(* PLC project Unnamed, Unknown Unnamed 1 *)
(* stored: creationDateTime 2023-10-18T21:45:43, modificationDateTime 2023-10-21T23:16:36 *)

PROGRAM program0
  VAR
    Emrg_Stop : BOOL;
    Output_switch : BOOL;
    change_filter : BOOL;
    Gray_water_level : INT;
    Filter_Input_water_level : INT;
    Filter_Output_water_level : INT;
    Clean_water_level : INT := 0;
    Graywater_Pump_RPM : INT;
    Filterwater_Pump_RPM : INT;
    Cleanwater_Pump_RPM : INT;
    Filterwater_Valve : BOOL;
    Cleanwater_Valve : BOOL;
    Filter_inflow_Valve : BOOL;
    Min_Water_Level : INT := 5;
    Max_Water_Level : INT := 25;
    Max_pump_speed : INT := 2000;
    Min_pump_speed : INT := 0;
    Mem1 : BOOL;
    Mem2 : BOOL;
    Mem3 : BOOL;
  END_VAR

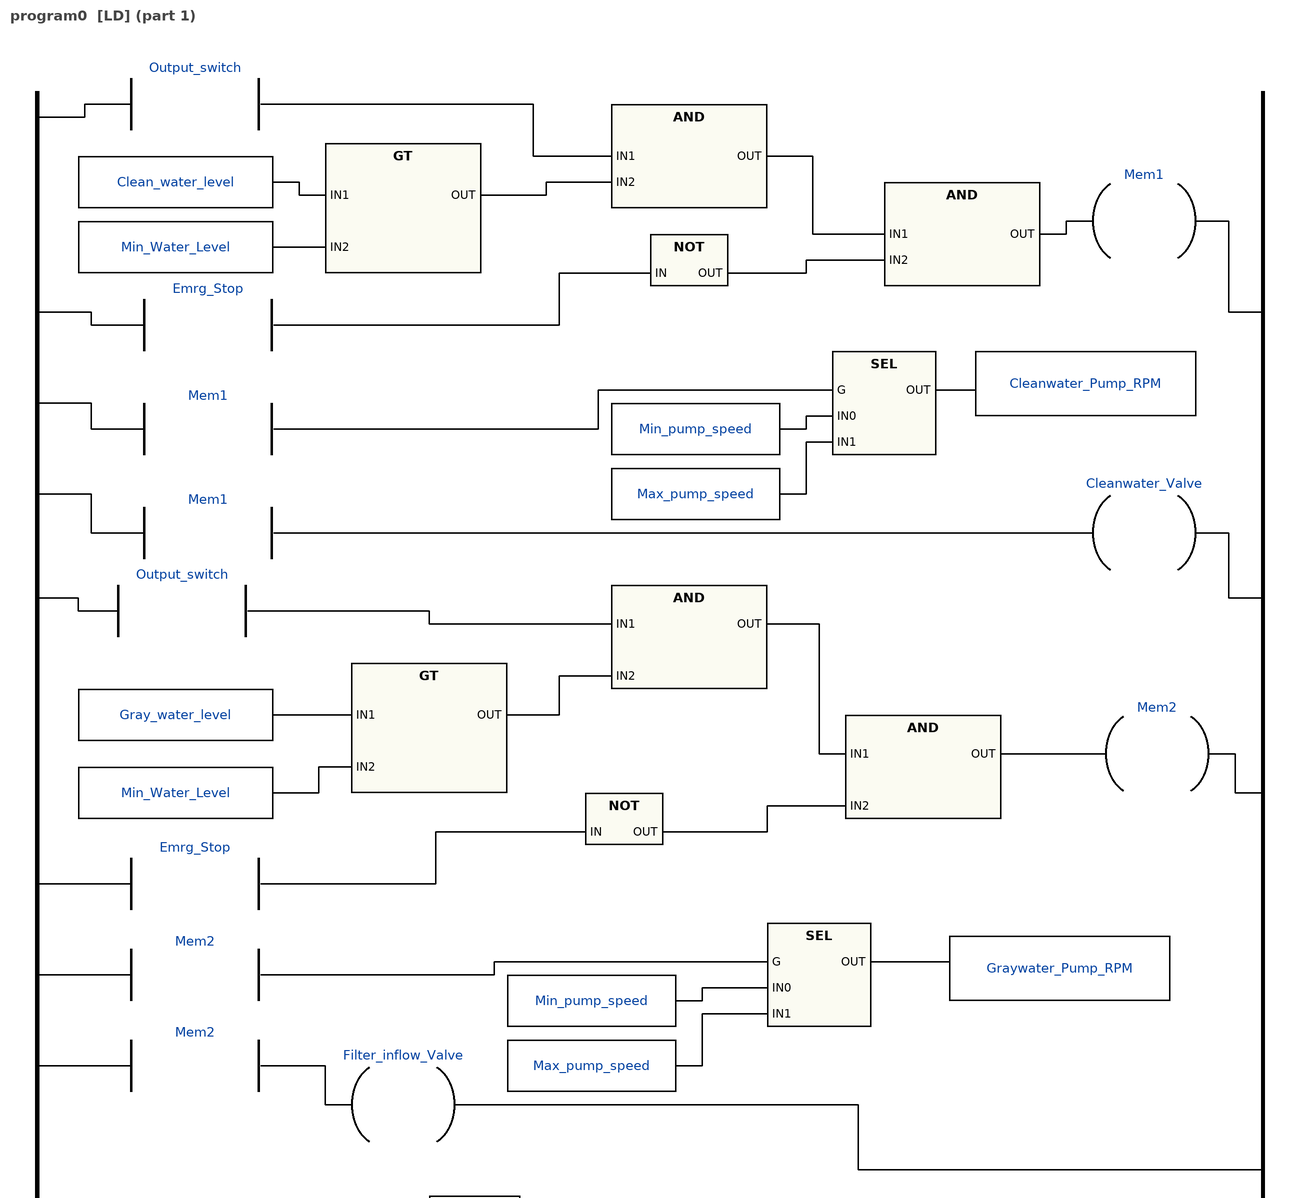
(* LD diagram, written out as Structured Text *)
Mem1 := Output_switch AND Clean_water_level > Min_Water_Level AND NOT Emrg_Stop;
Cleanwater_Pump_RPM := SEL(Mem1, Min_pump_speed, Max_pump_speed);
Cleanwater_Valve := Mem1;
Mem2 := Output_switch AND Gray_water_level > Min_Water_Level AND NOT Emrg_Stop;
Graywater_Pump_RPM := SEL(Mem2, Min_pump_speed, Max_pump_speed);
Filter_inflow_Valve := Mem2;
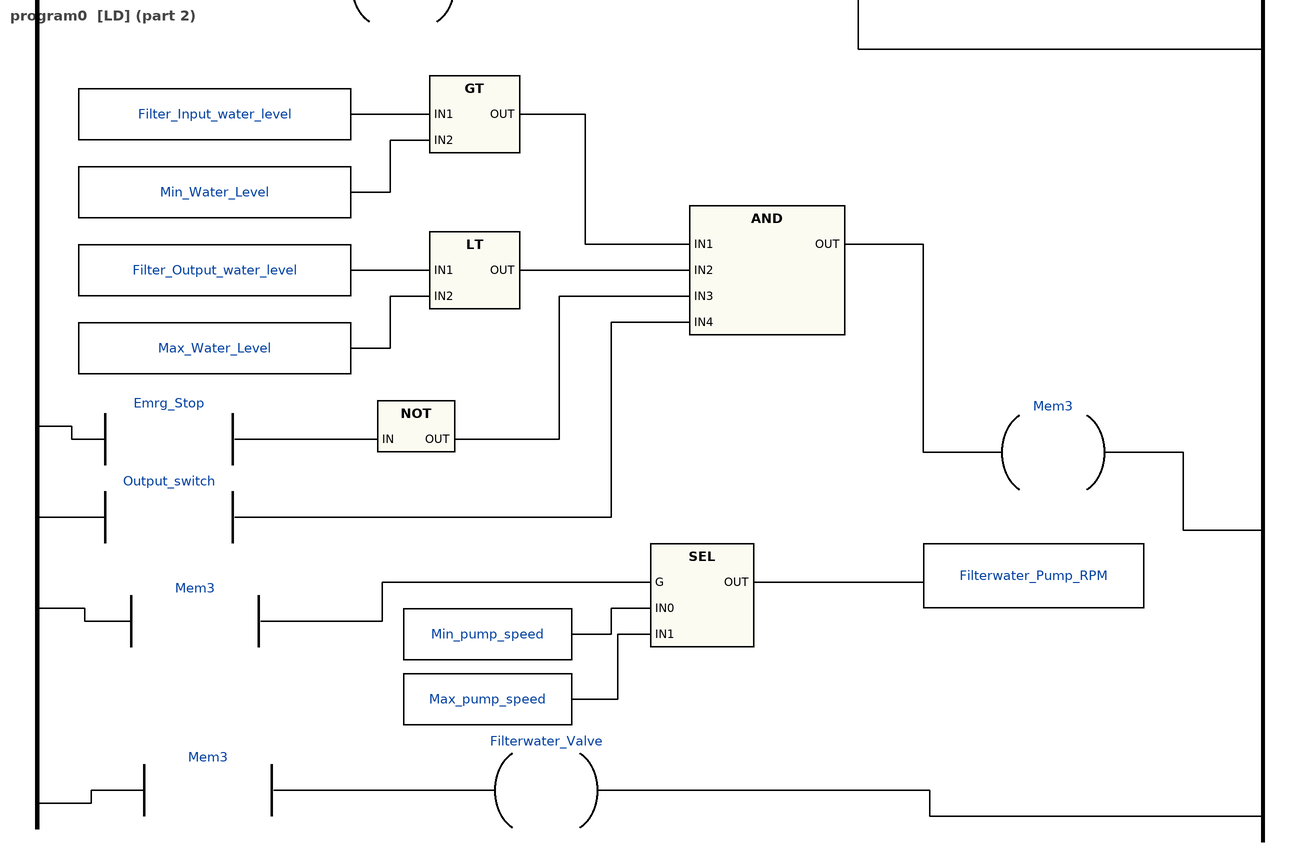
Mem3 := Filter_Input_water_level > Min_Water_Level AND Filter_Output_water_level < Max_Water_Level AND NOT Emrg_Stop AND Output_switch;
Filterwater_Pump_RPM := SEL(Mem3, Min_pump_speed, Max_pump_speed);
Filterwater_Valve := Mem3;
END_PROGRAM

CONFIGURATION Config0
  RESOURCE Res0 ON PLC
    TASK task0(INTERVAL := T#20ms, PRIORITY := 0);
    PROGRAM instance0 WITH task0 : program0;
  END_RESOURCE
END_CONFIGURATION
